INTERFACE I_HpAxis

END_INTERFACE

(* stored: Version 1.1.0.1, ProductVersion 3.1.4024.12
   Itf I_HpAxis: Id {709b750c-c769-44cd-9e1b-c9de775b9494} *)
